// TIA Portal V21 export
TYPE "Std_AllarmeDaUtenza"
   STRUCT
      Allarme : Bool;
      AllarmeSilenziato : Bool;
      Tipo : Bool;
      Indice : Bool;
   END_STRUCT;
END_TYPE
